// TIA Portal V20 export
FUNCTION_BLOCK "FB_ShuttleExt"   // FB59, SCL
{ S7_Optimized_Access := 'TRUE' }
// stored: MemoryReserve 100, SetENOAutomatically false
   VAR_INPUT
      iStartSeqCond : Bool;   // Start Sequence Conditions
      iJobReq : Bool;   // Job Request - From Main
      iIntGateOpened : Bool;   // Internal Gate Opened - From DI
      iIntGateClosed : Bool;   // Internal Gate Closed - From DI
      iExtGateOpened : Bool;   // External Gate Opened - From DI
      iExtGateClosed : Bool;   // External Gate Closed - From DI
      iShuttlePosInt : Bool;   // Shuttle Inside the Machine - Param
      iShuttlePosSas : Bool;   // Shuttle Inside the Sas - Param
      iShuttlePosExt : Bool;   // Shuttle Outside the Machine - Param
      iShuttlePosExtSetPoint : LReal;   // Shuttle Outside Position Setpoint - Param
      iShuttlePosSasSetPoint : LReal;   // Shuttle SasPosition Setpoint - Param
      iShuttleMoving : Bool;   // Shuttle is moving - From FB_LoaderAxis
      iShuttleInPos : Bool;   // Shuttle pos. reached - From FB_LoaderAxis
      iExtLoaderInSafePos : Bool;   // Gripper in Safe Position - Param
      iPLC_DateAndTime : DTL;
      iStepPause : Bool;
   END_VAR
   VAR_OUTPUT
      oExtGateOpenReq { ExternalAccessible := 'False'; ExternalVisible := 'False'; ExternalWritable := 'False'} : Bool;   // External Gate Opening Request - To DO
      oExtGateCloseReq { ExternalAccessible := 'False'; ExternalVisible := 'False'; ExternalWritable := 'False'} : Bool;   // External Gate Closing Request - To DO
      oIntGateOpenReq { ExternalAccessible := 'False'; ExternalVisible := 'False'; ExternalWritable := 'False'} : Bool;   // Internal Gate Opening Request - To DO
      oIntGateCloseReq { ExternalAccessible := 'False'; ExternalVisible := 'False'; ExternalWritable := 'False'} : Bool;   // Internal Gate Closing Request - To DO
      oShuttleStartReq { ExternalAccessible := 'False'; ExternalVisible := 'False'; ExternalWritable := 'False'} : Bool;   // Shuttle Start Order - To FB_LoaderAxis
      oShuttlePosSetPoint { ExternalAccessible := 'False'; ExternalVisible := 'False'; ExternalWritable := 'False'} : Real;   // Shuttle Position Setpoint - To FB_LoaderAxis
   END_VAR
   VAR
      sCurrent_Step_NB : Int;   // Active Step Number
      sCheck_Step_Condition : Bool;   // Check Step Condition
      sOneStepForward : Bool;
      sRTOneStepForward : R_TRIG;
      sOneStepMode { S7_SetPoint := 'True'} : Bool;
      sStepForward : Bool;
      sInterface : "UDT_SequenceInterface";   // Sequence Interface
      sExtGateOpenReq { ExternalAccessible := 'False'; ExternalVisible := 'False'; ExternalWritable := 'False'} : Bool;   // External Gate Opening Request
      sExtGateCloseReq { ExternalAccessible := 'False'; ExternalVisible := 'False'; ExternalWritable := 'False'} : Bool;   // External Gate Closing Request
      sIntGateOpenReq { ExternalAccessible := 'False'; ExternalVisible := 'False'; ExternalWritable := 'False'} : Bool;   // Internal Gate Opening Request
      sIntGateCloseReq { ExternalAccessible := 'False'; ExternalVisible := 'False'; ExternalWritable := 'False'} : Bool;   // Internal Gate Closing Request
      sShuttleStartReq { ExternalAccessible := 'False'; ExternalVisible := 'False'; ExternalWritable := 'False'} : Bool;   // Shuttle Start Request
      sShuttlePosSetPoint { ExternalAccessible := 'False'; ExternalVisible := 'False'; ExternalWritable := 'False'} : Real;   // Shuttle Position Setpoint
      sHistory : Struct
         Activation : Bool;
         Steps : Array[0..99] of Int;
         Date_Time : Array[0..99] of DTL;
      END_STRUCT;
      StepText : "FB_GetTextErrorCode";
   END_VAR
   VAR_TEMP
      tIndex : Int;   // Index
   END_VAR
   VAR CONSTANT
      S00_INIT : Int := 0;
      S10_CHECK_SHUTTLE_POSITION : Int := 10;
      S20_CLOSE_EXT_GATE : Int := 20;
      S30_OPEN_INT_GATE : Int := 30;
      S40_SHUTTLE_TO_SAS_START_REQ : Int := 40;
      S50_SHUTTLE_TO_SAS_POS_REACHED : Int := 50;
      S60_CLOSE_INT_GATE : Int := 60;
      S70_OPEN_EXT_GATE : Int := 70;
      S80_MOVE_SHUTTLE_TO_OUT_START_REQ : Int := 80;
      S90_MOVE_SHUTTLE_TO_OUT_POS_REACHED : Int := 90;
      S100_CLOSE_EXT_GATE : Int := 100;
      S195_JOB_DONE : Int := 195;
   END_VAR
   // StepText.sCode_error[0].ErrorCode := 0;
   // StepText.sCode_error[1].ErrorCode := 10;
   // StepText.sCode_error[2].ErrorCode := 20;
   // StepText.sCode_error[3].ErrorCode := 30;
   // StepText.sCode_error[4].ErrorCode := 40;
   // StepText.sCode_error[5].ErrorCode := 50;
   // StepText.sCode_error[6].ErrorCode := 60;
   // StepText.sCode_error[7].ErrorCode := 70;
   // StepText.sCode_error[8].ErrorCode := 80;
   // StepText.sCode_error[9].ErrorCode := 90;
   // StepText.sCode_error[10].ErrorCode := 95;
   // StepText.sCode_error[0].ErrorText := 'S00 : INIT';
   // StepText.sCode_error[1].ErrorText := 'S10 : CHECK SHUTTLE POSITION';
   // StepText.sCode_error[2].ErrorText := 'S20 : OPEN INT GATE';
   // StepText.sCode_error[3].ErrorText := 'S30 : SHUTTLE TO SAS START REQ';
   // StepText.sCode_error[4].ErrorText := 'S40 : SHUTTLE TO SAS POS REACHED';
   // StepText.sCode_error[5].ErrorText := 'S50 : CLOSE INT GATE';
   // StepText.sCode_error[6].ErrorText := 'S60 : OPEN EXT GATE';
   // StepText.sCode_error[7].ErrorText := 'S70 : MOVE SHUTTLE TO OUT START REQ';
   // StepText.sCode_error[8].ErrorText := 'S80 : MOVE SHUTTLE TO OUT POS REACHED';
   // StepText.sCode_error[9].ErrorText := 'S90 : CLOSE EXT GATE';
   // StepText.sCode_error[10].ErrorText := 'S95 : JOB DONE';
BEGIN
   REGION Description header 
       //==================================================================================
       // POSALUX Swiss SA / (C) Copyright 2025
       //----------------------------------------------------------------------------------
       // Title: FB_ShuttleExt
       // Comment/Function: 
       // Author: Fabien WALDT
       // Engineering: TIA Portal v17
       //----------------------------------------------------------------------------------
       // Change log table:
       // Version  | Date     | Expert in charge | Changes applied
       // ---------|----------|------------------|-----------------------------------------
       // 00.00.01 | 20250527 | WFA              | First released version
       // =================================================================================
   END_REGION

   REGION Define condition to start
       IF #iStartSeqCond THEN
           #sInterface.SequenceReleased := TRUE;
       ELSE
           // Standard sequencer controls
           #sInterface.SequenceReleased := FALSE;
           #sCurrent_Step_NB := #S00_INIT;
           #sInterface.SequenceRun := FALSE;
           #sInterface.JobDone := FALSE;
           #sCheck_Step_Condition := FALSE;

           // Dedicated sequencer controls
           #sExtGateOpenReq := FALSE;
           #sExtGateCloseReq := FALSE;
           #sIntGateOpenReq := FALSE;
           #sIntGateCloseReq := FALSE;
           #sShuttleStartReq := FALSE;
           #sShuttlePosSetPoint := 0.0;
           // Add specifics controls 
       END_IF;

       // Reset interface error
       IF #sInterface.Reset THEN
           #sInterface.Error := FALSE;
       END_IF;

       // Reset start when axis in position
       IF #iShuttleInPos THEN
           #sShuttleStartReq := FALSE;
       END_IF;

       // One step forward
       #sRTOneStepForward.CLK := #sOneStepForward;
       #sRTOneStepForward();
       #sStepForward := (NOT #sOneStepMode OR (#sOneStepMode AND #sRTOneStepForward.Q)) AND NOT #iStepPause;
       #sOneStepForward := FALSE;
   END_REGION

   REGION Sequence Function
       CASE #sCurrent_Step_NB OF
           #S00_INIT:
               REGION S00 INIT
                   #sCheck_Step_Condition := TRUE;
               END_REGION
           #S10_CHECK_SHUTTLE_POSITION:
               REGION S10_CHECK_SHUTTLE_POSITION
                   #sCheck_Step_Condition := TRUE;
               END_REGION
           #S20_CLOSE_EXT_GATE:
               REGION S20_CLOSE_EXT_GATE
                   #sExtGateOpenReq := FALSE;
                   #sExtGateCloseReq := TRUE;
                   #sCheck_Step_Condition := TRUE;
               END_REGION
           #S30_OPEN_INT_GATE:
               REGION S30_OPEN_INT_GATE
                   #sIntGateOpenReq := TRUE;
                   #sIntGateCloseReq := FALSE;
                   #sCheck_Step_Condition := TRUE;
               END_REGION
           #S40_SHUTTLE_TO_SAS_START_REQ:
               REGION S40_SHUTTLE_TO_SAS_START_REQ
                   #sShuttleStartReq := #iIntGateOpened AND NOT #iShuttlePosSas;
                   #sShuttlePosSetPoint := LREAL_TO_REAL(#iShuttlePosSasSetPoint);
                   #sCheck_Step_Condition := TRUE;
               END_REGION
           #S50_SHUTTLE_TO_SAS_POS_REACHED:
               REGION S50_SHUTTLE_TO_SAS_POS_REACHED
                   #sCheck_Step_Condition := TRUE;
               END_REGION
           #S60_CLOSE_INT_GATE:
               REGION S60_CLOSE_INT_GATE
                   #sIntGateOpenReq := FALSE;
                   #sIntGateCloseReq := TRUE;
                   #sCheck_Step_Condition := TRUE;
               END_REGION
           #S70_OPEN_EXT_GATE:
               REGION S70_OPEN_EXT_GATE
                   #sExtGateOpenReq := TRUE;
                   #sExtGateCloseReq := FALSE;
                   #sCheck_Step_Condition := TRUE;
               END_REGION
           #S80_MOVE_SHUTTLE_TO_OUT_START_REQ:
               REGION S80_MOVE_SHUTTLE_TO_OUT_START_REQ
                   #sShuttleStartReq := #iExtGateOpened AND NOT #iShuttlePosExt;
                   #sShuttlePosSetPoint := LREAL_TO_REAL(#iShuttlePosExtSetPoint);
                   #sCheck_Step_Condition := TRUE;
               END_REGION
           #S90_MOVE_SHUTTLE_TO_OUT_POS_REACHED:
               REGION S90_MOVE_SHUTTLE_TO_OUT_POS_REACHED
                   #sCheck_Step_Condition := TRUE;
               END_REGION
           #S100_CLOSE_EXT_GATE:
               REGION S100_CLOSE_EXT_GATE
                   #sIntGateOpenReq := FALSE;
                   #sIntGateCloseReq := TRUE;
                   #sExtGateOpenReq := FALSE;
                   #sExtGateCloseReq := TRUE;
                   #sCheck_Step_Condition := TRUE;
               END_REGION
           #S195_JOB_DONE:
               REGION S195_JOB_DONE
                   #sInterface.JobDone := TRUE;
                   #sCheck_Step_Condition := TRUE;
               END_REGION
           ELSE:
               #sInterface.Error := TRUE;
       END_CASE;
   END_REGION

   REGION Sequence Next Step Condition
       IF #sCheck_Step_Condition THEN
           CASE #sCurrent_Step_NB OF
               #S00_INIT:
                   REGION S00 INIT
                       IF #sInterface.SequenceReleased AND #iJobReq THEN
                           #sCurrent_Step_NB := #S10_CHECK_SHUTTLE_POSITION;
                           #sInterface.SequenceRun := TRUE;
                           #sCheck_Step_Condition := FALSE;
                       ELSE
                           #sInterface.SequenceRun := FALSE;
                       END_IF;
                   END_REGION
               #S10_CHECK_SHUTTLE_POSITION:
                   REGION S10_CHECK_SHUTTLE_POSITION
                       IF #sInterface.SequenceReleased AND #sStepForward AND #iShuttlePosInt THEN
                           #sCurrent_Step_NB := #S20_CLOSE_EXT_GATE;
                           #sCheck_Step_Condition := FALSE;
                       ELSIF #sInterface.SequenceReleased AND #sStepForward AND #iShuttlePosSas THEN
                           #sCurrent_Step_NB := #S60_CLOSE_INT_GATE;
                           #sCheck_Step_Condition := FALSE;
                       ELSIF #sInterface.SequenceReleased AND #sStepForward AND #iShuttlePosExt THEN
                           #sCurrent_Step_NB := #S100_CLOSE_EXT_GATE;
                           #sCheck_Step_Condition := FALSE;
                       END_IF;
                   END_REGION
               #S20_CLOSE_EXT_GATE:
                   REGION S20_CLOSE_EXT_GATE
                       IF #sInterface.SequenceReleased AND #sStepForward AND #iExtGateClosed THEN
                           #sCurrent_Step_NB := #S30_OPEN_INT_GATE;
                           #sCheck_Step_Condition := FALSE;
                       END_IF;
                   END_REGION
               #S30_OPEN_INT_GATE:
                   REGION S30_OPEN_INT_GATE
                       IF #sInterface.SequenceReleased AND #sStepForward AND #iIntGateOpened THEN
                           #sCurrent_Step_NB := #S40_SHUTTLE_TO_SAS_START_REQ;
                           #sCheck_Step_Condition := FALSE;
                       END_IF;
                   END_REGION
               #S40_SHUTTLE_TO_SAS_START_REQ:
                   REGION S40_SHUTTLE_TO_SAS_START_REQ
                     //  IF #sInterface.SequenceReleased AND #sStepForward AND (#ShuttleMoving OR #ShuttlePosSas) THEN
                       IF #sInterface.SequenceReleased AND (#iShuttleMoving OR #iShuttlePosSas) THEN
                           #sCurrent_Step_NB := #S50_SHUTTLE_TO_SAS_POS_REACHED;
                           #sCheck_Step_Condition := FALSE;
                       END_IF;
                   END_REGION
               #S50_SHUTTLE_TO_SAS_POS_REACHED:
                   REGION S50_SHUTTLE_TO_SAS_POS_REACHED
                       IF #sInterface.SequenceReleased AND #sStepForward AND NOT #sShuttleStartReq AND #iShuttlePosSas THEN
                           #sCurrent_Step_NB := #S60_CLOSE_INT_GATE;
                           #sCheck_Step_Condition := FALSE;
                       END_IF;
                   END_REGION
               #S60_CLOSE_INT_GATE:
                   REGION S60_CLOSE_INT_GATE
                       IF #sInterface.SequenceReleased AND #sStepForward AND #iIntGateClosed THEN
                           #sCurrent_Step_NB := #S70_OPEN_EXT_GATE;
                           #sCheck_Step_Condition := FALSE;
                       END_IF;
                   END_REGION
               #S70_OPEN_EXT_GATE:
                   REGION S70_OPEN_EXT_GATE
                       IF #sInterface.SequenceReleased AND #sStepForward AND #iExtGateOpened THEN
                           #sCurrent_Step_NB := #S80_MOVE_SHUTTLE_TO_OUT_START_REQ;
                           #sCheck_Step_Condition := FALSE;
                       END_IF;
                   END_REGION
               #S80_MOVE_SHUTTLE_TO_OUT_START_REQ:
                   REGION S80_MOVE_SHUTTLE_TO_OUT_START_REQ
                       IF #sInterface.SequenceReleased AND (#iShuttleMoving OR #iShuttlePosExt) THEN
                           #sCurrent_Step_NB := #S90_MOVE_SHUTTLE_TO_OUT_POS_REACHED;
                           #sCheck_Step_Condition := FALSE;
                       END_IF;
                   END_REGION
               #S90_MOVE_SHUTTLE_TO_OUT_POS_REACHED:
                   REGION S90_MOVE_SHUTTLE_TO_OUT_POS_REACHED
                       IF #sInterface.SequenceReleased AND #sStepForward AND NOT #sShuttleStartReq AND #iShuttlePosExt THEN
                           #sCurrent_Step_NB := #S100_CLOSE_EXT_GATE;
                           #sCheck_Step_Condition := FALSE;
                       END_IF;
                   END_REGION
               #S100_CLOSE_EXT_GATE:
                   REGION S100_CLOSE_EXT_GATE
                       IF #sInterface.SequenceReleased AND #sStepForward AND #iIntGateClosed AND #iExtGateClosed THEN
                           #sCurrent_Step_NB := #S195_JOB_DONE;
                           #sCheck_Step_Condition := FALSE;
                       END_IF;
                   END_REGION
               #S195_JOB_DONE:
                   REGION S195_JOB_DONE
                       IF NOT #iJobReq THEN
                           #sCurrent_Step_NB := #S00_INIT;
                           #sCheck_Step_Condition := FALSE;
                           #sInterface.JobDone := FALSE;
                       END_IF;
                   END_REGION
               ELSE
                   #sInterface.Error := TRUE;
           END_CASE;
       END_IF;
   END_REGION

   REGION Outputs Update
       #oExtGateOpenReq  := #sExtGateOpenReq;
       #oExtGateCloseReq := #sExtGateCloseReq;
       #oIntGateOpenReq  := #sIntGateOpenReq;
       #oIntGateCloseReq := #sIntGateCloseReq;
       #oShuttleStartReq:= #sShuttleStartReq AND ((#iShuttlePosExt AND #iExtLoaderInSafePos) OR NOT #iShuttlePosExt);
       #oShuttlePosSetPoint:= #sShuttlePosSetPoint;
   END_REGION

   REGION Steps - Date and Time History
       IF #sHistory.Activation THEN
           IF #sHistory.Steps[0] <> #sCurrent_Step_NB THEN
               FOR #tIndex := 98 TO 0 BY -1 DO
                   #sHistory.Steps[#tIndex + 1] := #sHistory.Steps[#tIndex];
                   #sHistory.Date_Time[#tIndex + 1] := #sHistory.Date_Time[#tIndex];
               END_FOR;
               #sHistory.Steps[0] := #sCurrent_Step_NB;
               #sHistory.Date_Time[0] := #iPLC_DateAndTime;
           END_IF;
       END_IF;
   END_REGION

   REGION Steps Text
       #StepText(iErrorCode := #sCurrent_Step_NB,
                 oErrorText => #StepText.oErrorText);
   END_REGION
END_FUNCTION_BLOCK
